TYPE DUT_HMI_General_Manuals :
STRUCT
	PS : ARRAY[0..CNC.NUM_MAX_MANUALS_GENERAL-1] OF BOOL;
	LS : ARRAY[0..CNC.NUM_MAX_MANUALS_GENERAL-1] OF BOOL;
END_STRUCT
END_TYPE

(* stored: Version 1.1.0.1, ProductVersion 3.1.4024.13
   DUT DUT_HMI_General_Manuals: Id {065e2469-fe21-4c60-a64f-53002e5b48e2} *)
